ABB RAPID module: MainModule.mod

MODULE MainModule
    !***********************************************************
    Func robtarget SoundToPosition(num i,num SoundArrayMiddle2{*,*})
        VAR robtarget PositionIntermediate;
        VAR num Excursion;
        !Read from file
        !Open "Home:/default.txt",FilePosition;!wait to change
        !SoundData:=ReadNum(FilePosition);
        IF SoundArrayMiddle2{i,3}<0 OR SoundArrayMiddle2{i,3}>7 THEN
            ErrWrite "Wrong Note","out of octave"\RL2:="please check input array";
            stop;
        ENDIF
        IF (SoundArrayMiddle2{i,2}<0) and (SoundArrayMiddle2{i,3}=1 or SoundArrayMiddle2{i,3}=4) THEN
            ErrWrite "Wrong Note","inexist black button"\RL2:="please check input array";
            stop;
        ELSEIF (SoundArrayMiddle2{i,2}>0) and (SoundArrayMiddle2{i,3}=7 or SoundArrayMiddle2{i,3}=3) THEN
            ErrWrite "Wrong Note","inexist black button"\RL2:="please check input array";
            stop;
        ENDIF
        Excursion:=ButtonLength*(7*(SoundArrayMiddle2{i,1}-4)+SoundArrayMiddle2{i,3}-1+SoundArrayMiddle2{i,2}/2);
        IF abs(Excursion)>55 THEN
            ErrWrite "out of range of motion","cannot get close to this point"\RL2:="please check input array";
            stop;
        ENDIF
        PositionIntermediate:=offs(pCenter,abs(SoundArrayMiddle2{i,2})*(-BlackToWhite),Excursion,0);
        RETURN PositionIntermediate;
    ENDFUNC

    !Func num CalcTime(VAR robtarget TargetPositionIntermediate,VAR num Speed)
    !VAR robtarget CurrentPositionIntermediate;
    !CurrentPositionIntermediate:=CRobT();
    !MoveTime:=Abs(TargetPositionIntermediate.trans.x-CurrentPositionIntermediate.trans.x)/Speed;!unit:1s
    !RETURN MoveTime;
    !ENDFUNC

    PROC Play(num SoundArrayMiddle1{*,*})
        FOR i FROM 1 TO Dim(SoundArrayMiddle1,1) DO
            TargetPosition:=SoundToPosition(i,SoundArrayMiddle1);
            !TimeToWait:=CurrentSoundTime-CalcTime(TargetPosition,GlobalSpeed);
            ClkReset clock1;
            ClkStart clock1;
            MoveJ TargetPosition,vmax,fine,Tool0;
            TimeToWait:=CurrentSoundTime-ClkRead(clock1)-0.323;
            !unit:1s
            MoveL Offs(TargetPosition,0,0,-PressDepth),vmax,fine,Tool0;
            IF TimeToWait>0 THEN
                WaitTime TimeToWait;
            ELSE
                ErrWrite\I,"timepoint late","";
            ENDIF
            MoveL TargetPosition,vmax,fine,Tool0;
        ENDFOR
    ENDPROC

    PROC TCP_Socket()
        SocketClose client_socket;
        SocketCreate client_socket;
        SocketConnect client_socket,"127.0.0.1",8080;
        TPWrite "Socket client connect successful";
        SocketSend client_socket\Str:="This is robot";
        SocketReceive client_socket\Str:=received_string;
        InputProcess;
    ENDPROC

    Proc InputProcess()
        start:=0;
        default_val:=1;
        FOR i FROM 1 TO 3 DO
            start:=found+1;
            found:=StrFind(received_string,start,";");
            default_val:=found-start;
            sTOn_True:=strtoval(StrPart(received_string,start,default_val),InputProcessStringArray{i});
            IF sTOn_True THEN
                TPWrite ""\Num:=InputProcessStringArray{i};
            ELSE
                TPWrite "InputProcessStringArray error!";
            ENDIF
        ENDFOR
        start:=0;
        default_val:=1;
        FOR i FROM 1 TO 3 DO
            FOR j FROM 1 TO 3 DO
                start:=found+1;
                found:=StrFind(received_string,start,",");
                default_val:=found-start;
                sTOn_True:=strtoval(StrPart(InputProcessStringArray{i},start,default_val),SoundArray{i,j});
                IF sTOn_True THEN
                    TPWrite ""\Num:=SoundArray{i,j};
                ELSE
                    TPWrite "SoundArray error!";
                ENDIF
            ENDFOR
        ENDFOR
    ENDPROC

    PROC main()
        !MoveAbsJ Home,v1000,z50,Tool0;
        MoveL pHome,v300,fine,Tool0;
        MoveL pCenterAbove,v300,fine,Tool0;
        Play(SoundArray);
        MoveL pCenterAbove,v300,fine,Tool0;
        MoveL pHome,v300,fine,Tool0;
    ENDPROC

ENDMODULE
